TYPE ST_CycleDataCSV :
STRUCT
    uiNestId            : UINT;
    sGeneralResult      : STRING(20);
    sSiliconeResult     : STRING(20);
    sFlippingResult     : STRING(20);
    sDate               : STRING(255);
    sTime               : STRING(255);
END_STRUCT
END_TYPE

(* stored: Version 1.1.0.1, ProductVersion 3.1.4026.18
   DUT ST_CycleDataCSV: Id {bc9fe13d-b510-4993-a490-82d8860bdcaf} *)
